(* CODESYS project Timer_count.project

Project tree, tasks and I/O mapping:
  Drive : Unidrive M400, Nidec Control Techniques, version 1.8.0.9
    application Application
      Task Configuration
        Freewheeling
      program Freewheeling [ST]: MAin
      Custom Menu
      global variables M30
      function block hrs_count [ST]
    <Empty>
  Advanced Link Editor
*)

// Drive/Application/M30
(* This file is auto-generated by the system. Any changes maybe lost.  Please do not change this file.*)
{attribute 'qualified_only'}
VAR_GLOBAL

// Parameter Number 1. Mode(s)  OpenLoop  RFC-A  RFC-S  Regen .
 
 //working_time_hrs 

//
{attribute 'get_access' := 'ReadUserParameterDINT(0, 30, 1)'}
{attribute 'get_bitaccess' := 'ReadUserParameterBit(0, 30, 1, BITNR)'}
{attribute 'set_bitaccess' := 'WriteUserParameterBit(0, 30, 1, Working_time, BITNR)'}
{attribute 'set_access' := 'WriteUserParameterDINT(0, 30, 1, Working_time)'}
{attribute 'monitoring_instead' := 'ReadUserParameterDINT(0, 30, 1)'}
Working_time : DINT;

END_VAR

// Drive/Application/Freewheeling
PROGRAM Freewheeling  //v1.0.1 Jul 11/2019
VAR		
	hrs_count_0		: hrs_count; // FB declaration
	wrt_ms			: DINT;  //working time ms
	wrt_seg			: DINT;	 //working time seg
	wrt_min			: DINT;  //working time min
	wrt_hrs			: DINT;	 //working time hrs
	mins_completed	: BOOL;  //setup min completed
	segs_completed	: BOOL;  //setup seg completed
	hrs_completed	: BOOL;  //setup hrs completed
	hrs_to_count    : DINT;  //hrs to count
END_VAR

IF M20.P024 <2 THEN                         //Minimun hours to count= 2 
	M20.P024:=2;
END_IF

IF M20.P024 >480 THEN                      //  maximun time to count 480hrs =20 days   
	M20.P024:=480;
END_IF

hrs_to_count    := M20.P024;                     

MAin();                                          //call main FB
M18.P011		:= BOOL_TO_INT(segs_completed);  //Completed seconds
M18.P012		:= BOOL_TO_INT(mins_completed);  //Completed minutes
M18.P013		:= BOOL_TO_INT(hrs_completed);   //Completed hours

M20.P021		:= wrt_seg;    					// accumulated seconds counts                   
M20.P022		:= wrt_min;   					// accumulated minutes counts
M20.P023		:= wrt_hrs;	  					//accumulated HRS counts

ACTION MAin:
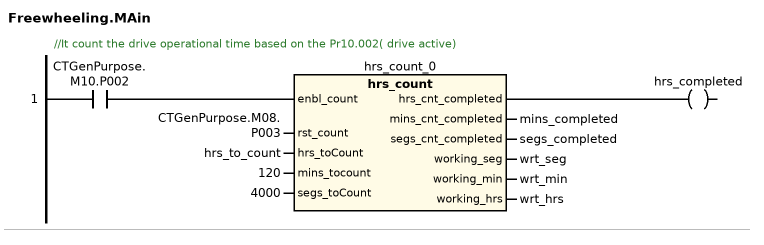
// NETWORK 1
// //It count the drive operational time based on the Pr10.002( drive active)
hrs_count_0(
    enbl_count := CTGenPurpose.M10.P002,
    rst_count := CTGenPurpose.M08.P003,
    hrs_toCount := hrs_to_count,
    mins_tocount := 120,
    segs_toCount := 4000,
    mins_cnt_completed => mins_completed,
    segs_cnt_completed => segs_completed,
    working_seg => wrt_seg,
    working_min => wrt_min,
    working_hrs => wrt_hrs); // hrs_count
hrs_completed := hrs_count_0.hrs_cnt_completed;
END_ACTION

END_PROGRAM

// Drive/Application/hrs_count
 // this function block count time when enable input is TRUE, the runing time is stored in non volatile variable "DINT" so the time wont be lost when drive is off.
 //
FUNCTION_BLOCK hrs_count
VAR_INPUT
	enbl_count				:BOOL	:=	FALSE;  //Enables counting
	rst_count 				:BOOL	:=	FALSE;  //Reset accumulated count
	hrs_toCount 			:DINT;              // Hours to count  ( It only activate the output  hrs_cnt_completed)
	mins_tocount  			:DINT;              //Minutes to count ( it oly activate mins_cnt_completed)
	segs_toCount			:DINT;				//Seconds to count ( it oly activate segs_cnt_completed)
END_VAR	
VAR_OUTPUT
	hrs_cnt_completed		:BOOL;
	mins_cnt_completed		:BOOL;
	segs_cnt_completed		:BOOL;		
	working_seg				:DINT;
	working_min				:DINT;
	working_hrs 			:DINT;
	
END_VAR
VAR
	last_enbl_count_status 	: BOOL;
	flag					: BOOL := TRUE;
	captured_time			: TIME;
	running					: TIME;
	working_ms				: DINT;
	init					: BOOL := TRUE;
	working_ms2				: DINT;
	flag1					: BOOL;
	
END_VAR

IF init =TRUE THEN 
	working_ms2 	:=M30.Working_time;      	//When drives power up Update the stored working time
	init			:=FALSE;                 	//Only once making  init=false 
END_IF

IF hrs_toCount <2 THEN                         //Minimun hours to count= 2 
	hrs_toCount:=2;
END_IF

IF hrs_toCount >480 THEN                      //  maximun time to count 480hrs =20 days   
	hrs_toCount:=480;
END_IF

IF mins_toCount <5 THEN                         //Minimun minutes to count= 5 minutos  
	mins_toCount:=5;
END_IF

IF mins_toCount >28800 THEN                      // Max time to count 28800 minutes = 20 days    
	mins_toCount:=28800;
END_IF

IF enbl_count <> last_enbl_count_status THEN   // To detect is the status change of the  counting DI 
	IF (enbl_count = TRUE AND flag ) THEN      // If the change was from False to  true  enable the flag to start counting time
		captured_time 	:= TIME();
		flag			:= FALSE;
		flag1			:= TRUE;
	END_IF
	IF (enbl_count=FALSE AND flag1) THEN		//Si el cambio es de true a falso 
		working_ms2 	:=M30.Working_time; 
		flag1			:=FALSE;
		flag			:=TRUE;
		running 		:=T#0MS;
	END_IF
END_IF
last_enbl_count_status:= enbl_count;

IF  NOT flag THEN
	running	:=TIME()-captured_time;
END_IF

working_ms	:= TIME_TO_DINT(running)+working_ms2;

working_seg := working_ms/1000;
working_min := working_ms/60000;
working_hrs := working_ms/3600000;
M30.Working_time:=working_ms;
   

IF (working_seg>=segs_toCount) THEN
	segs_cnt_completed:=TRUE;
END_IF
IF (working_min>=mins_toCount) THEN
	mins_cnt_completed:=TRUE;
END_IF
IF (working_hrs>=hrs_toCount) THEN
	hrs_cnt_completed:=TRUE;
END_IF

IF rst_count THEN                      //reset all 
	working_ms			:=0;
	working_ms2			:=0;
	working_seg     	:=0;
	working_min			:=0;	
	M30.Working_time	:=0;
	hrs_cnt_completed	:=FALSE;
	mins_cnt_completed  :=FALSE;
	segs_cnt_completed	:=FALSE;
END_IF

END_FUNCTION_BLOCK
